PROGRAM Read_FatigueCam
VAR
	fbEL6001		: FB_FatigueCam;
	RxBufferPcCom	: ComBuffer;	
	TxBufferPcCom	: ComBuffer;
	
	Timer	: TON;
	i		: INT := 60;
	
	fbTime 		: FB_LocalSystemTime := ( bEnable := TRUE, dwCycle := 1 );
	bValid		: BOOL := FALSE;
	TimeStr		: STRING;
	
	Year		: USINT;
	Month		: USINT;
	bDate		: USINT;
	Hour		: USINT;
	Minute		: USINT;
	Second		: USINT;
	
	YearBin		: STRING;
	MonthBin	: STRING;
	bDateBin	: STRING;
	HourBin		: STRING;
	MinuteBin	: STRING;
	SecondBin	: STRING;
	
	BinStr		: ARRAY [1..4] OF STRING;
	TimeBin		: STRING;
	
	//Command		: LINT := 16#DE1527378DAA;
	//Command		: LINT := 16#000000008CAA;
	Command			: ULINT := 16#00;
	Response		: STRING := 'ABC';
	EventID			: STRING := '00';
	prevEventID		: STRING;
	EventCode		: STRING;
END_VAR

(* sync time every 1 minute *)
IF i = 60 THEN 
	(*
	WHILE bValid = FALSE DO //wait until time sync
		fbTime(bValid => bValid);
	END_WHILE
	*)
	
	IF bValid = FALSE THEN //wait until time sync
		fbTime(bValid => bValid);
	END_IF
	
	TimeStr		:= SYSTEMTIME_TO_STRING(fbTime.systemTime); //get datetime
	//TimeStr		:= '2013-12-19-17:23:30.000';
	Year		:= STRING_TO_USINT(MID(STR := TimeStr, LEN := 2, POS := 3));
	Month		:= STRING_TO_USINT(MID(STR := TimeStr, LEN := 2, POS := 6));
	bDate		:= STRING_TO_USINT(MID(STR := TimeStr, LEN := 2, POS := 9));
	Hour		:= STRING_TO_USINT(MID(STR := TimeStr, LEN := 2, POS := 12));
	Minute		:= STRING_TO_USINT(MID(STR := TimeStr, LEN := 2, POS := 15));
	Second		:= STRING_TO_USINT(MID(STR := TimeStr, LEN := 2, POS := 18));
	
	(* convert datetime to binary *)
	YearBin		:= BYTE_TO_BINSTR(in := Year, iPrecision := 6);
	MonthBin	:= BYTE_TO_BINSTR(in := Month, iPrecision := 4);
	bDateBin	:= BYTE_TO_BINSTR(in := bDate, iPrecision := 5);
	HourBin		:= BYTE_TO_BINSTR(in := Hour, iPrecision := 5);
	MinuteBin	:= BYTE_TO_BINSTR(in := Minute, iPrecision := 6);
	SecondBin	:= BYTE_TO_BINSTR(in := Second, iPrecision := 6);
	BinStr[4]	:= CONCAT(YearBin, MonthBin); 
	BinStr[4]	:= CONCAT(BinStr[4], bDateBin);
	BinStr[4]	:= CONCAT(BinStr[4], HourBin); 
	BinStr[4]	:= CONCAT(BinStr[4], MinuteBin);
	BinStr[4]	:= CONCAT(BinStr[4], SecondBin);
	
	(* separate bytes *)
	BinStr[1]	:= LEFT(STR := BinStr[4], SIZE := 8);
	BinStr[2]	:= MID(STR := BinStr[4], LEN := 8, POS := 9);
	BinStr[3]	:= MID(STR := BinStr[4], LEN := 8, POS := 17);
	BinStr[4]	:= RIGHT(STR := BinStr[4], SIZE := 8);
	
	(* build sync command *)
	TimeBin		:= CONCAT('2#', BinStr[4]);
	TimeBin		:= CONCAT(TimeBin, BinStr[3]);
	TimeBin		:= CONCAT(TimeBin, BinStr[2]);
	TimeBin		:= CONCAT(TimeBin, BinStr[1]);
	TimeBin		:= CONCAT(TimeBin, '10001101'); //8D
	TimeBin		:= CONCAT(TimeBin, '10101010'); //AA
	Command		:= STRING_TO_ULINT(TimeBin);
	//Command		:= 16#DE1527378DAA;
	
	(* send sync command *)
	WHILE Response <> LWORD_TO_HEXSTR(in := command, iPrecision := 1, bLoCase := FALSE) DO
		fbEL6001(
			TxBuffer	:= GVL.TxBufferEL, 
			RxBuffer	:= GVL.RxBufferEL,
			Command		:= Command,
			Response	=> Response
		);
	END_WHILE
	i := 0;
END_IF

(* fatigue cam request event *)
Command	:= 16#000000008CAA;
Timer(IN := FALSE);
fbEL6001(
	TxBuffer	:= GVL.TxBufferEL, 
	RxBuffer	:= GVL.RxBufferEL,
	Command		:= Command,
	EventID		=> EventID,
	EventCode	=> EventCode,
	Response	=> Response,
);
	
//IF EventCode = '0' OR EventID = prevEventID THEN
IF EventCode = '' OR EventID = prevEventID THEN
	EventCode 	:= '0';
	//EventID	:= '';
ELSE
	prevEventID	:= EventID;
END_IF
i := i+1;

END_PROGRAM

(* stored: Version 1.1.0.1, ProductVersion 3.1.4024.6
   POU Read_FatigueCam: Id {aef089b1-c7c5-479f-8336-a7bf9b8b2785}, SpecialFunc None *)
